PROGRAM PRG_SampleVisitor
VAR
	fbExporter					: FB_Visitor;
	fbElementA					: FB_ElementA;
	fbElementB					: FB_ElementB;	

	bEnable						:BOOL;
END_VAR

//*************************************************************
// Disable Test enviroment
//*************************************************************	
	IF NOT bEnable THEN
		
		RETURN;
		
	END_IF
	
//*************************************************************
// Call Objects
//*************************************************************
	fbElementA.accept(fbExporter);
	fbElementB.accept(fbExporter);

END_PROGRAM

(* stored: Version 1.1.0.1
   POU PRG_SampleVisitor: Id {fff20f15-e1aa-48b0-81e8-cf63c8903751}, SpecialFunc None *)
